FUNCTION_BLOCK Recipe_10015_DoubleChocoCookie
VAR_INPUT
	TaskID	: 	LREAL;
	Execute :	BOOL;
END_VAR
VAR_OUTPUT
	Recipedone : BOOL;
	RecipeInfo	: DUT_RECIPEOFFER;
	InitDone	: BOOL;
END_VAR
VAR
	Done	: BOOL;
	
END_VAR

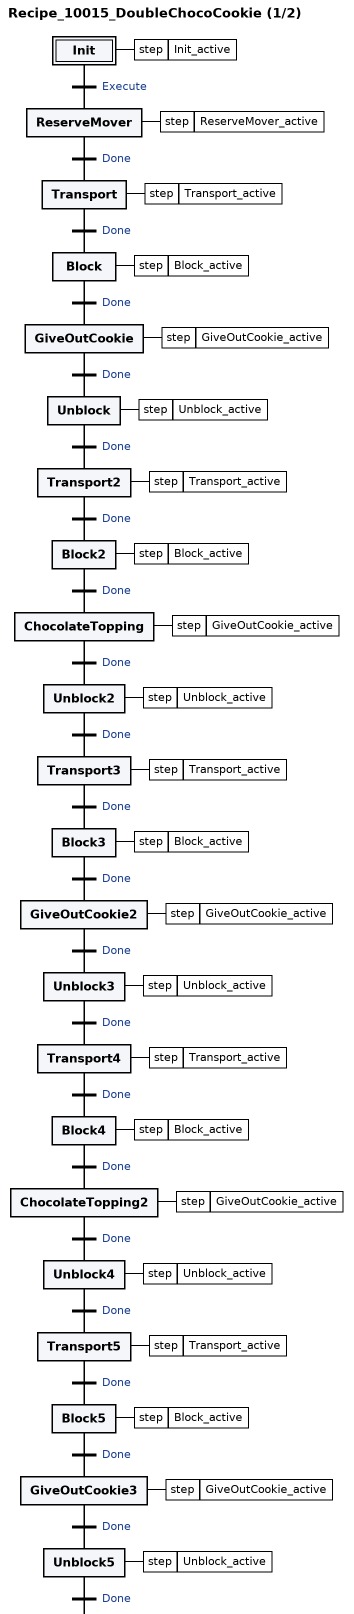
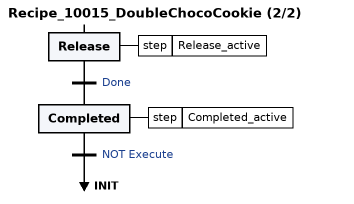
INITIAL_STEP Init:
    Init_active(N);  // step action
END_STEP
TRANSITION FROM Init TO ReserveMover
    := Execute;
END_TRANSITION
STEP ReserveMover:
    ReserveMover_active(N);  // step action
END_STEP
TRANSITION FROM ReserveMover TO Transport
    := Done;
END_TRANSITION
STEP Transport:
    Transport_active(N);  // step action
END_STEP
TRANSITION FROM Transport TO Block
    := Done;
END_TRANSITION
STEP Block:
    Block_active(N);  // step action
END_STEP
TRANSITION FROM Block TO GiveOutCookie
    := Done;
END_TRANSITION
STEP GiveOutCookie:
    GiveOutCookie_active(N);  // step action
END_STEP
TRANSITION FROM GiveOutCookie TO Unblock
    := Done;
END_TRANSITION
STEP Unblock:
    Unblock_active(N);  // step action
END_STEP
TRANSITION FROM Unblock TO Transport2
    := Done;
END_TRANSITION
STEP Transport2:
    Transport_active(N);  // step action
END_STEP
TRANSITION FROM Transport2 TO Block2
    := Done;
END_TRANSITION
STEP Block2:
    Block_active(N);  // step action
END_STEP
TRANSITION FROM Block2 TO ChocolateTopping
    := Done;
END_TRANSITION
STEP ChocolateTopping:
    GiveOutCookie_active(N);  // step action
END_STEP
TRANSITION FROM ChocolateTopping TO Unblock2
    := Done;
END_TRANSITION
STEP Unblock2:
    Unblock_active(N);  // step action
END_STEP
TRANSITION FROM Unblock2 TO Transport3
    := Done;
END_TRANSITION
STEP Transport3:
    Transport_active(N);  // step action
END_STEP
TRANSITION FROM Transport3 TO Block3
    := Done;
END_TRANSITION
STEP Block3:
    Block_active(N);  // step action
END_STEP
TRANSITION FROM Block3 TO GiveOutCookie2
    := Done;
END_TRANSITION
STEP GiveOutCookie2:
    GiveOutCookie_active(N);  // step action
END_STEP
TRANSITION FROM GiveOutCookie2 TO Unblock3
    := Done;
END_TRANSITION
STEP Unblock3:
    Unblock_active(N);  // step action
END_STEP
TRANSITION FROM Unblock3 TO Transport4
    := Done;
END_TRANSITION
STEP Transport4:
    Transport_active(N);  // step action
END_STEP
TRANSITION FROM Transport4 TO Block4
    := Done;
END_TRANSITION
STEP Block4:
    Block_active(N);  // step action
END_STEP
TRANSITION FROM Block4 TO ChocolateTopping2
    := Done;
END_TRANSITION
STEP ChocolateTopping2:
    GiveOutCookie_active(N);  // step action
END_STEP
TRANSITION FROM ChocolateTopping2 TO Unblock4
    := Done;
END_TRANSITION
STEP Unblock4:
    Unblock_active(N);  // step action
END_STEP
TRANSITION FROM Unblock4 TO Transport5
    := Done;
END_TRANSITION
STEP Transport5:
    Transport_active(N);  // step action
END_STEP
TRANSITION FROM Transport5 TO Block5
    := Done;
END_TRANSITION
STEP Block5:
    Block_active(N);  // step action
END_STEP
TRANSITION FROM Block5 TO GiveOutCookie3
    := Done;
END_TRANSITION
STEP GiveOutCookie3:
    GiveOutCookie_active(N);  // step action
END_STEP
TRANSITION FROM GiveOutCookie3 TO Unblock5
    := Done;
END_TRANSITION
STEP Unblock5:
    Unblock_active(N);  // step action
END_STEP
TRANSITION FROM Unblock5 TO Release
    := Done;
END_TRANSITION
STEP Release:
    Release_active(N);  // step action
END_STEP
TRANSITION FROM Release TO Completed
    := Done;
END_TRANSITION
STEP Completed:
    Completed_active(N);  // step action
END_STEP
TRANSITION FROM Completed TO INIT
    := NOT Execute;
END_TRANSITION

ACTION GiveOutCookie_active:
Done := FALSE;

ExecuteSkill.SkillID 			:= 1210;
ExecuteSkill.SkillName	 		:= 'Dispense Chocolate Topping';
ExecuteSkill.Parameter[1].ID 	:= 1;
ExecuteSkill.Parameter[1].Name 	:= 'Amount';
ExecuteSkill.Parameter[1].Value := 5.31;
ExecuteSkill();
Done := TRUE;
END_ACTION

ACTION Unblock_active:
Done := FALSE;

//Skill auswählen
ExecuteSkill.SkillID := 1316;
ExecuteSkill.SkillName	 := 'Unblock Mover';

//Parameter setzen
ExecuteSkill.Parameter[1].ID := 1;
ExecuteSkill.Parameter[1].Name := 'TaskID';
ExecuteSkill.Parameter[1].Value := TaskID;

//Skill hinzufügen
ExecuteSkill();


Done := TRUE;
END_ACTION

ACTION Release_active:
Done := FALSE;


ExecuteSkill.SkillID 			:= 1311;
ExecuteSkill.SkillName	 		:= 'Release Mover';
ExecuteSkill.Parameter[1].ID 	:= 1;
ExecuteSkill.Parameter[1].Name 	:= 'TaskID';
ExecuteSkill.Parameter[1].Value := TaskID;
ExecuteSkill();

Done := TRUE;
END_ACTION

ACTION Init_active:
RecipeDone := FALSE;



// Initialisation of Recipe Parameters an name etc
RecipeInfo.Name := 'Double Chocolate Cookie';
RecipeInfo.Description := 'This Recipe produces a simple, but still delicious two-layer Cookie with Chocolate inside';
RecipeInfo.Dummy := FALSE;
RecipeInfo.RecipeID := 10015;

Initdone := TRUE;
//Parameter 1:
(*
	RecipeInfo.UserParameter[1].Dummy 		:= 
	RecipeInfo.UserParameter[1].Default		:=
	RecipeInfo.UserParameter[1].Description	:=
	RecipeInfo.UserParameter[1].MaxValue	:=
	RecipeInfo.UserParameter[1].MinValue	:=
	RecipeInfo.UserParameter[1].Name		:=
	RecipeInfo.UserParameter[1].Unit		:=
*)
//Parameter 2:

(*
	RecipeInfo.UserParameter[2].Dummy 		:= 
	RecipeInfo.UserParameter[2].Default		:=
	RecipeInfo.UserParameter[2].Description	:=
	RecipeInfo.UserParameter[2].MaxValue	:=
	RecipeInfo.UserParameter[2].MinValue	:=
	RecipeInfo.UserParameter[2].Name		:=
	RecipeInfo.UserParameter[2].Unit		:=
*)

//Parameter 3:

(*
	RecipeInfo.UserParameter[3].Dummy 		:= 
	RecipeInfo.UserParameter[3].Default		:=
	RecipeInfo.UserParameter[3].Description	:=
	RecipeInfo.UserParameter[3].MaxValue	:=
	RecipeInfo.UserParameter[3].MinValue	:=
	RecipeInfo.UserParameter[3].Name		:=
	RecipeInfo.UserParameter[3].Unit		:=
*)

//Parameter 4:

(*
	RecipeInfo.UserParameter[4].Dummy 		:= 
	RecipeInfo.UserParameter[4].Default		:=
	RecipeInfo.UserParameter[4].Description	:=
	RecipeInfo.UserParameter[4].MaxValue	:=
	RecipeInfo.UserParameter[4].MinValue	:=
	RecipeInfo.UserParameter[4].Name		:=
	RecipeInfo.UserParameter[4].Unit		:=
*)


//Parameter 5:

(*
	RecipeInfo.UserParameter[5].Dummy 		:= 
	RecipeInfo.UserParameter[5].Default		:=
	RecipeInfo.UserParameter[5].Description	:=
	RecipeInfo.UserParameter[5].MaxValue	:=
	RecipeInfo.UserParameter[5].MinValue	:=
	RecipeInfo.UserParameter[5].Name		:=
	RecipeInfo.UserParameter[5].Unit		:=
*)
END_ACTION

ACTION Completed_active:
RecipeDone := TRUE;
Done := FALSE;
END_ACTION

ACTION Transport_active:
Done := FALSE;

//Skill auswählen
ExecuteSkill.SkillID 		:= 1320;
ExecuteSkill.SkillName	 	:= 'Transport Mover';

//Geschwindigkeit setzen
ExecuteSkill.Parameter[1].ID := 3;
ExecuteSkill.Parameter[1].Name := 'Velocity';
ExecuteSkill.Parameter[1].Value := 3000;


ExecuteSkill();
Done := TRUE;
END_ACTION

ACTION Done_active:
Done := TRUE;
END_ACTION

ACTION ReserveMover_active:
Done := FALSE;


ExecuteSkill.SkillID := 1310;
ExecuteSkill.SkillName	 := 'Reserve Mover';
ExecuteSkill.Parameter[1].ID := 1;
ExecuteSkill.Parameter[1].Name := 'TaskID';
ExecuteSkill.Parameter[1].Value := TaskID;
ExecuteSkill();

Done := TRUE;
END_ACTION

ACTION Block_active:
Done := FALSE;

//Skill auswählen
ExecuteSkill.SkillID := 1315;
ExecuteSkill.SkillName	 := 'Block Mover';

//Parameter setzen
ExecuteSkill.Parameter[1].ID := 1;
ExecuteSkill.Parameter[1].Name := 'TaskID';
ExecuteSkill.Parameter[1].Value := TaskID;

//Skill hinzufügen
ExecuteSkill();


Done := TRUE;
END_ACTION

END_FUNCTION_BLOCK

(* stored: Version 1.1.0.1, ProductVersion 3.1.0.25
   POU Recipe_10015_DoubleChocoCookie: Id {b29ec41f-43ab-479a-a131-818f4c95622a}
   Action GiveOutCookie_active: Id {064af2de-4c9b-48fe-8b7f-f1c2dbcef051}
   Action Unblock_active: Id {24503286-7558-45fd-96b5-c1193f78e2f2}
   Action Release_active: Id {2e035cc7-9b20-4508-b3d2-90899af3bdc8}
   Action Init_active: Id {336883c9-b268-44dc-8246-cb4e2504bc43}
   Action Completed_active: Id {9238b342-afa0-464e-a62f-99d430bdb25a}
   Action Transport_active: Id {941776fa-95ed-4bbd-a912-a1d50a87535d}
   Action Done_active: Id {c678d82c-0bd9-4590-a097-379f0c82b291}
   Action ReserveMover_active: Id {f02393f2-e873-45eb-bf70-fb1ed8f2428f}
   Action Block_active: Id {f4898579-f515-4d64-8b98-ff53345814c7} *)
